(* POU FB_BACnet_RemoteProgram, ST *)
FUNCTION_BLOCK FB_BACnet_RemoteProgram
VAR_IN_OUT
	RemoteDevice		: FB_BACnet_RemoteDevice;
END_VAR
VAR_OUTPUT
	bReady				: BOOL;
	ePrgState			: E_BACNETPROGRAMSTATE;
	ePrgReasonHalt		: E_BACNETPROGRAMERROR;
	bOverridden			: BOOL;
	bOutOfService		: BOOL;
	bFault				: BOOL;
	bInAlarm			: BOOL;
	bError				: BOOL;
	nErrorId			: UINT;
END_VAR
VAR
	_ProgramState AT%I*: WORD;			(* ~(BACnet_ProgramState 				:		: )
								   			(BACnet_ObjectType 					: PROG	: )
			                            	(BACnet_RemoteCycletimeRead 		: 1000	: )
											(BACnet_RemoteFlagsRead        		: 1    	: )
                                   			(BACnet_RemoteResubscriptionInterval: 240 	: )
	                                		(BACnet_RemoteCycleTimeWrite   		: 1000	: )
	                                		(BACnet_RemoteFlagsWrite       		: 1		: )	*)
	_ReasonForHalt AT%I*: WORD;			(* ~(BACnet_ReasonForHalt 				: 		: )	*)
	_StatusFlags AT%I*: WORD;			(* ~(BACnet_StatusFlags 				:		: )	*)
	_nUpdateCount : UDINT := 0;
	_StatusFlagsBits : ST_BACnet_StatusFlags;
END_VAR
(* update client device *)
IF RemoteDevice._nUpdateCount = _nUpdateCount THEN
	RemoteDevice();
END_IF
(* remind current number of update counter *)
_nUpdateCount := RemoteDevice._nUpdateCount;

IF RemoteDevice.bFirstCycle THEN
	(* first call of the server device since reboot/reset *)
	bReady := FALSE;

ELSIF NOT RemoteDevice.bOperational THEN
	nErrorId := BACnet_ERR_OPERATIONAL;
	bReady := FALSE;

ELSIF _StatusFlags >= 4 THEN
	(* clear error flag *)
	nErrorId := BACnet_ERR_NO_ERROR;

	(* ready state *)
	bReady := TRUE;

	(* decode status flags *)
	_StatusFlagsBits := F_BACnet_StatusFlags(_StatusFlags);

	(* copy states to output *)
	bOverridden := _StatusFlagsBits.overridden;
	bOutOfService := _StatusFlagsBits.out_of_service;
	bFault := _StatusFlagsBits.fault;
	bInAlarm := _StatusFlagsBits.in_alarm;

	(* present value from BACnet *)
	ePrgState := _ProgramState;

	(* other states *)
	ePrgReasonHalt := _ReasonForHalt;
ELSE
	(* server device not ready, reset local ready also *)
	bReady := FALSE;
	(* and set error ID *)
	nErrorId := BACnet_ERR_WRONG_MAPPING;
END_IF

(* set error flag *)
bError := (nErrorId <> BACnet_ERR_NO_ERROR);
END_FUNCTION_BLOCK

(* POU FB_BACnet_RemoteProgram_EX, ST *)
FUNCTION_BLOCK FB_BACnet_RemoteProgram_EX
VAR_INPUT
	bEnablePV			: BOOL;
	ePV					: E_BACNETPROGRAMREQUEST;
	bRetrigger			: BOOL; (* execute selected request on raising edge again *)
END_VAR
VAR_IN_OUT
	RemoteDevice		: FB_BACnet_RemoteDevice;
END_VAR
VAR_OUTPUT
	bReady				: BOOL;
	ePrgState			: E_BACNETPROGRAMSTATE;
	ePrgChangeReq		: E_BACNETPROGRAMREQUEST;
	ePrgReasonHalt		: E_BACNETPROGRAMERROR;
	bOverridden			: BOOL;
	bOutOfService		: BOOL;
	bFault				: BOOL;
	bInAlarm			: BOOL;
	bProcessError		: BOOL;
	bOtherFault			: BOOL;
	tObjectID		: DINT := -1;
	bError				: BOOL;
	nErrorId			: UINT;
END_VAR
VAR
	_ProgramState AT%I*: WORD;			(* ~(BACnet_ProgramState 				:		: )
											(BACnet_ObjectType 					: PROG	: )
											(BACnet_RemoteCycletimeRead 		: 1000	: )
											(BACnet_RemoteFlagsRead        		: 1    	: )
											(BACnet_RemoteResubscriptionInterval: 240 	: )
											(BACnet_RemoteCycleTimeWrite   		: 1000	: )
											(BACnet_RemoteFlagsWrite       		: 1		: )	*)
	_ProgramChangeState AT%I*: WORD;	(* ~(BACnet_ProgramChange 				:		: )	*)
	_ReasonForHalt AT%I*: WORD;			(* ~(BACnet_ReasonForHalt 				: 		: )	*)
	_StatusFlags AT%I*: WORD;			(* ~(BACnet_StatusFlags 				:		: )	*)
	_Reliability AT%I*: WORD;			(* ~(BACnet_Reliability 				:		: )	*)
	_ProgramChangeRequest AT%Q*: WORD;	(* ~(BACnet_ProgramChange 				:		: )	*)
	_ObjectId AT%I*: DWORD;				(* ~(BACnet_ObjectIdentifier			:		: LINK) *)
	_nUpdateCount : UDINT := 0;
	_StatusFlagsBits : ST_BACnet_StatusFlags;
	_rtrigRetriggerPv : R_TRIG;
END_VAR
(* update client device *)
IF RemoteDevice._nUpdateCount = _nUpdateCount THEN
	RemoteDevice();
END_IF
(* remind current number of update counter *)
_nUpdateCount := RemoteDevice._nUpdateCount;

(* call trigger *)
_rtrigRetriggerPv(CLK:= bRetrigger, Q=> );

IF RemoteDevice.bFirstCycle THEN
	(* first call of the server device since reboot/reset *)
	bReady := FALSE;
	_ProgramChangeRequest := 0;
ELSIF NOT RemoteDevice.bOperational THEN
	nErrorId := BACnet_ERR_OPERATIONAL;
	bReady := FALSE;

ELSIF (F_BACnet_GetObjType(_ObjectId) <> BACnetObjectType_Program) THEN
	(* wrong mapping / invalid object ID *)
	IF _ObjectId = 0 THEN
		nErrorId := BACnet_ERR_WRONG_MAPPING;
	ELSE
		nErrorId := BACnet_ERR_INVALID_OBJECTID;
	END_IF
	bReady := FALSE;
	tObjectID := 16#FFFFFFFF;

ELSIF _StatusFlags >= 4 THEN
	(* clear error flag *)
	nErrorId := BACnet_ERR_NO_ERROR;

	(* ready state *)
	bReady := TRUE;

	(* decode status flags *)
	_StatusFlagsBits := F_BACnet_StatusFlags(_StatusFlags);

	(* copy states to output *)
	bOverridden := _StatusFlagsBits.overridden;
	bOutOfService := _StatusFlagsBits.out_of_service;
	bFault := _StatusFlagsBits.fault;
	bInAlarm := _StatusFlagsBits.in_alarm;
	bProcessError := (_Reliability = BACnetReliability_process_error);
	bOtherFault := (_Reliability = BACnetReliability_unreliable_other);
	tObjectID := _ObjectId;

	(* present value from BACnet *)
	ePrgState := _ProgramState;
	(* present value to BACnet *)
	IF bEnablePV THEN
		IF _rtrigRetriggerPv.Q THEN
			(* trigger request *)
			_ProgramChangeRequest := 0;
		ELSE
			(* set request value *)
			_ProgramChangeRequest := ePV;
		END_IF
	ELSE
		_ProgramChangeRequest := 0;
	END_IF
	(* other states *)
	ePrgReasonHalt := _ReasonForHalt;
	ePrgChangeReq := _ProgramChangeState;

ELSE
	(* server device not ready, reset local ready also *)
	bReady := FALSE;
	(* and set error ID *)
	nErrorId := BACnet_ERR_WRONG_MAPPING;
END_IF

(* set error flag *)
bError := (nErrorId <> BACnet_ERR_NO_ERROR);
END_FUNCTION_BLOCK

(* POU FB_BACnet_RemoteProgram_WR, ST *)
FUNCTION_BLOCK FB_BACnet_RemoteProgram_WR
VAR_INPUT
	bEnablePV			: BOOL;
	ePV					: E_BACNETPROGRAMREQUEST;
	bRetrigger			: BOOL; (* execute selected request on raising edge again *)
END_VAR
VAR_IN_OUT
	RemoteDevice		: FB_BACnet_RemoteDevice;
END_VAR
VAR_OUTPUT
	bReady				: BOOL;
	ePrgState			: E_BACNETPROGRAMSTATE;
	ePrgReasonHalt		: E_BACNETPROGRAMERROR;
	bOverridden			: BOOL;
	bOutOfService		: BOOL;
	bFault				: BOOL;
	bInAlarm			: BOOL;
	bError				: BOOL;
	nErrorId			: UINT;
END_VAR
VAR
	_ProgramState AT%I*: WORD;			(* ~(BACnet_ProgramState 				:		: )
								   			(BACnet_ObjectType 					: PROG	: )
			                            	(BACnet_RemoteCycletimeRead 		: 1000	: )
											(BACnet_RemoteFlagsRead        		: 1    	: )
                                   			(BACnet_RemoteResubscriptionInterval: 240 	: )
	                                		(BACnet_RemoteCycleTimeWrite   		: 1000	: )
	                                		(BACnet_RemoteFlagsWrite       		: 1		: )	*)
	_ReasonForHalt AT%I*: WORD;			(* ~(BACnet_ReasonForHalt 				: 		: )	*)
	_StatusFlags AT%I*: WORD;			(* ~(BACnet_StatusFlags 				:		: )	*)
	_ProgramChangeRequest AT%Q*: WORD;	(* ~(BACnet_ProgramChange 				:		: )	*)
	_nUpdateCount : UDINT := 0;
	_StatusFlagsBits : ST_BACnet_StatusFlags;
	_rtrigRetriggerPv : R_TRIG;
END_VAR
(* update client device *)
IF RemoteDevice._nUpdateCount = _nUpdateCount THEN
	RemoteDevice();
END_IF
(* remind current number of update counter *)
_nUpdateCount := RemoteDevice._nUpdateCount;

(* call trigger *)
_rtrigRetriggerPv(CLK:= bRetrigger, Q=> );

IF RemoteDevice.bFirstCycle THEN
	(* first call of the server device since reboot/reset *)
	bReady := FALSE;
	_ProgramChangeRequest := 0;
ELSIF NOT RemoteDevice.bOperational THEN
	nErrorId := BACnet_ERR_OPERATIONAL;
	bReady := FALSE;

ELSIF _StatusFlags >= 4 THEN
	(* clear error flag *)
	nErrorId := BACnet_ERR_NO_ERROR;

	(* ready state *)
	bReady := TRUE;

	(* decode status flags *)
	_StatusFlagsBits := F_BACnet_StatusFlags(_StatusFlags);

	(* copy states to output *)
	bOverridden := _StatusFlagsBits.overridden;
	bOutOfService := _StatusFlagsBits.out_of_service;
	bFault := _StatusFlagsBits.fault;
	bInAlarm := _StatusFlagsBits.in_alarm;

	(* present value from BACnet *)
	ePrgState := _ProgramState;
	(* present value to BACnet *)
	IF bEnablePV THEN
		IF _rtrigRetriggerPv.Q THEN
			(* trigger request *)
			_ProgramChangeRequest := 0;
		ELSE
			(* set request value *)
			_ProgramChangeRequest := ePV;
		END_IF
	ELSE
		_ProgramChangeRequest := 0;
	END_IF
	(* other states *)
	ePrgReasonHalt := _ReasonForHalt;
ELSE
	(* server device not ready, reset local ready also *)
	bReady := FALSE;
	(* and set error ID *)
	nErrorId := BACnet_ERR_WRONG_MAPPING;
END_IF

(* set error flag *)
bError := (nErrorId <> BACnet_ERR_NO_ERROR);
END_FUNCTION_BLOCK

(* POU FB_BACnet_RemotePulseConverter, ST *)
FUNCTION_BLOCK FB_BACnet_RemotePulseConverter
VAR_IN_OUT
	RemoteDevice		: FB_BACnet_RemoteDevice;
END_VAR
VAR_OUTPUT
	bReady				: BOOL;
	bOverridden			: BOOL;
	bOutOfService		: BOOL;
	bFault				: BOOL;
	bInAlarm			: BOOL;
	bError				: BOOL;
	nErrorId			: UINT;
END_VAR
VAR
	_StatusFlags AT%I*: UINT;		(* ~(BACnet_StatusFlags 				:		: )
										(BACnet_ObjectType 					: PC	: )
										(BACnet_RemoteCycletimeRead 		: 1000	: )
										(BACnet_RemoteFlagsRead        		: 1		: )
										(BACnet_RemoteResubscriptionInterval: 240	: )
                                		(BACnet_RemoteCycleTimeWrite   		: 1000	: )
                                		(BACnet_RemoteFlagsWrite       		: 1		: )	*)
	_StatusFlagsBits : ST_BACnet_StatusFlags;
	_nUpdateCount : UDINT := 0;
END_VAR
(* update client device *)
IF RemoteDevice._nUpdateCount = _nUpdateCount THEN
	RemoteDevice();
END_IF
(* remind current number of update counter *)
_nUpdateCount := RemoteDevice._nUpdateCount;

IF NOT RemoteDevice.bOperational THEN
	nErrorId := BACnet_ERR_OPERATIONAL;
	bReady := FALSE;

ELSIF _StatusFlags >= 4 THEN
	(* clear error flag *)
	nErrorId := BACnet_ERR_NO_ERROR;
	(* ready state *)
	bReady := TRUE;

	(* build bit states *)
	_StatusFlagsBits := F_BACnet_StatusFlags(_StatusFlags);

	(* copy states to output *)
	bOverridden := _StatusFlagsBits.overridden;
	bOutOfService := _StatusFlagsBits.out_of_service;
	bFault := _StatusFlagsBits.fault;
	bInAlarm := _StatusFlagsBits.in_alarm;

ELSE
	(* server device not ready, reset local ready also *)
	bReady := FALSE;
	(* and set error ID *)
	nErrorId := BACnet_ERR_WRONG_MAPPING;
END_IF

(* set error flag *)
bError := (nErrorId <> BACnet_ERR_NO_ERROR);
END_FUNCTION_BLOCK

(* POU FB_BACnet_RemotePulseConverter_EX, ST *)
FUNCTION_BLOCK FB_BACnet_RemotePulseConverter_EX
VAR_IN_OUT
	RemoteDevice	: FB_BACnet_RemoteDevice;
END_VAR
VAR_OUTPUT
	bReady			: BOOL;
	fPresentValue	: REAL;
	nCount			: UDINT;
	bOverridden		: BOOL;
	bOutOfService	: BOOL;
	bFault			: BOOL;
	bInAlarm		: BOOL;
	bOverRange		: BOOL;
	bUnderRange		: BOOL;
	bNoSensor		: BOOL;
	bOpenLoop		: BOOL;
	bShortedLoop	: BOOL;
	bCommFailure	: BOOL;
	bConfigError	: BOOL;
	bOtherFault		: BOOL;
	tObjectID		: T_BACnet_ObjectIdentifier := 16#FFFFFFFF;
	bError			: BOOL;
	nErrorId		: UINT;
END_VAR
VAR
	_ObjectId AT%I*: DWORD;		(* ~(BACnet_ObjectIdentifier			:		: LINK) *)
	_Count AT%I*: UDINT;		(* ~(BACnet_Count		 				:		: ) *)
	_PresentValue AT%I*: REAL;	(* ~(BACnet_PresentValue 				:		: )	*)
	_StatusFlags AT%I*: UINT;	(* ~(BACnet_StatusFlags 				:		: )
									(BACnet_ObjectType 					: PC	: )
									(BACnet_RemoteCycletimeRead 		: 1000	: )
									(BACnet_RemoteFlagsRead        		: 1		: )
									(BACnet_RemoteResubscriptionInterval: 240	: )
                                	(BACnet_RemoteCycleTimeWrite   		: 1000	: )
                                	(BACnet_RemoteFlagsWrite       		: 1		: )	*)
	_Reliability AT%I*:WORD;	(* ~(BACnet_Reliability					:		: )	*)
	_StatusFlagsBits : ST_BACnet_StatusFlags;
	_nUpdateCount : UDINT := 0;
END_VAR
(* update client device *)
IF RemoteDevice._nUpdateCount = _nUpdateCount THEN
	RemoteDevice();
END_IF
(* remind current number of update counter *)
_nUpdateCount := RemoteDevice._nUpdateCount;

IF NOT RemoteDevice.bOperational THEN
	nErrorId := BACnet_ERR_OPERATIONAL;
	bReady := FALSE;

ELSIF (F_BACnet_GetObjType(_ObjectId) <> BACnetObjectType_PulseConverter) THEN
	(* wrong mapping / invalid object ID *)
	IF _ObjectId = 0 THEN
		nErrorId := BACnet_ERR_WRONG_MAPPING;
	ELSE
		nErrorId := BACnet_ERR_INVALID_OBJECTID;
	END_IF
	bReady := FALSE;
	tObjectID := 16#FFFFFFFF;

ELSIF _StatusFlags >= 4 THEN
	(* clear error flag *)
	nErrorId := BACnet_ERR_NO_ERROR;
	(* ready state *)
	bReady := TRUE;

	(* present value *)
	fPresentValue := _PresentValue;
	nCount := _Count;

	(* build bit states *)
	_StatusFlagsBits := F_BACnet_StatusFlags(_StatusFlags);

	(* copy states to output *)
	bOverridden := _StatusFlagsBits.overridden;
	bOutOfService := _StatusFlagsBits.out_of_service;
	bFault := _StatusFlagsBits.fault;
	bInAlarm := _StatusFlagsBits.in_alarm;
	tObjectID := _ObjectId;

	(* reliability *)
	bOverRange	:= (_Reliability = BACnetReliability_over_range);
	bUnderRange	:= (_Reliability = BACnetReliability_under_range);
	bNoSensor	:= (_Reliability = BACnetReliability_no_sensor);
	bOpenLoop	:= (_Reliability = BACnetReliability_open_loop);
	bShortedLoop:= (_Reliability = BACnetReliability_shorted_loop);
	bCommFailure := (_Reliability = BACnetReliability_communication_failure);
	bConfigError:= (_Reliability = BACnetReliability_configuration_error);
	bOtherFault	:= (_Reliability = BACnetReliability_unreliable_other);

ELSE
	(* server device not ready, reset local ready also *)
	bReady := FALSE;
	(* and set error ID *)
	nErrorId := BACnet_ERR_WRONG_MAPPING;
END_IF

(* set error flag *)
bError := (nErrorId <> BACnet_ERR_NO_ERROR);
END_FUNCTION_BLOCK

(* POU FB_BACnet_RemoteSchedule, ST *)
FUNCTION_BLOCK FB_BACnet_RemoteSchedule
VAR_IN_OUT
	RemoteDevice			: FB_BACnet_RemoteDevice;
END_VAR
VAR_OUTPUT
	bReady				: BOOL;
	bPresentValue		: BOOL;
	bOverridden			: BOOL;
	bOutOfService		: BOOL;
	bFault				: BOOL;
	bInAlarm			: BOOL;
	bError				: BOOL;
	nErrorId			: UINT;
END_VAR
VAR
	_StatusFlags AT%I*: WORD; 	(* ~(BACnet_StatusFlags 				:		: )	*)
	_PresentValue AT%I*: BOOL;	(* ~(BACnet_PresentValueBool 			:		: )
									(BACnet_ObjectType 					: SCHED	: )
									(BACnet_RemoteCycletimeRead 		: 1000	: )
									(BACnet_RemoteFlagsRead        		: 1		: )
									(BACnet_RemoteResubscriptionInterval: 240	: )
                            		(BACnet_RemoteCycleTimeWrite   		: 1000	: )
                            		(BACnet_RemoteFlagsWrite       		: 1		: )	*)
	_StatusFlagsBits : ST_BACnet_StatusFlags;
	_nUpdateCount : UDINT := 0;
END_VAR
(* update client device *)
IF RemoteDevice._nUpdateCount = _nUpdateCount THEN
	RemoteDevice();
END_IF
(* remind current number of update counter *)
_nUpdateCount := RemoteDevice._nUpdateCount;

IF NOT RemoteDevice.bOperational THEN
	nErrorId := BACnet_ERR_OPERATIONAL;
	bReady := FALSE;

ELSIF _StatusFlags >= 4 THEN
	(* clear error flag *)
	nErrorId := BACnet_ERR_NO_ERROR;
	(* ready state *)
	bReady := TRUE;

	(* present value *)
	bPresentValue := _PresentValue;

	(* build bit states *)
	_StatusFlagsBits := F_BACnet_StatusFlags(_StatusFlags);

	(* copy states to output *)
	bOverridden := _StatusFlagsBits.overridden;
	bOutOfService := _StatusFlagsBits.out_of_service;
	bFault := _StatusFlagsBits.fault;
	bInAlarm := _StatusFlagsBits.in_alarm;

ELSE
	bReady := FALSE;
	(* and set error ID *)
	nErrorId := BACnet_ERR_WRONG_MAPPING;
END_IF

(* set error flag *)
bError := (nErrorId <> BACnet_ERR_NO_ERROR);
END_FUNCTION_BLOCK

(* POU FB_BACnet_RemoteSchedule_EX, ST *)
FUNCTION_BLOCK FB_BACnet_RemoteSchedule_EX
VAR_IN_OUT
	RemoteDevice			: FB_BACnet_RemoteDevice;
END_VAR
VAR_OUTPUT
	bReady				: BOOL;
	bPresentValue		: BOOL;
	bOverridden			: BOOL;
	bOutOfService		: BOOL;
	bFault				: BOOL;
	bInAlarm			: BOOL;
	bConfigError		: BOOL;
	bOtherFault			: BOOL;
	tObjectID			: T_BACnet_ObjectIdentifier := 16#FFFFFFFF;
	bError				: BOOL;
	nErrorId			: UINT;
END_VAR
VAR
	_ObjectId AT%I*: DWORD;				(* ~(BACnet_ObjectIdentifier			:		: LINK) *)
	_Reliability AT%I*: WORD; 			(* ~(BACnet_Reliability 				:		: )	*)
	_StatusFlags AT%I*: WORD; 			(* ~(BACnet_StatusFlags 				:		: )	*)
	_PresentValue AT%I*: BOOL;			(* ~(BACnet_PresentValueBool 			:		: )
											(BACnet_ObjectType 					: SCHED	: )
											(BACnet_RemoteCycletimeRead 		: 1000	: )
											(BACnet_RemoteFlagsRead        		: 1		: )
											(BACnet_RemoteResubscriptionInterval: 240	: )
                            				(BACnet_RemoteCycleTimeWrite   		: 1000	: )
                            				(BACnet_RemoteFlagsWrite       		: 1		: )	*)
	_StatusFlagsBits : ST_BACnet_StatusFlags;
	_nUpdateCount : UDINT := 0;
END_VAR
(* update client device *)
IF RemoteDevice._nUpdateCount = _nUpdateCount THEN
	RemoteDevice();
END_IF
(* remind current number of update counter *)
_nUpdateCount := RemoteDevice._nUpdateCount;

IF NOT RemoteDevice.bOperational THEN
	nErrorId := BACnet_ERR_OPERATIONAL;
	bReady := FALSE;

ELSIF (F_BACnet_GetObjType(_ObjectId) <> BACnetObjectType_Schedule) THEN
	(* wrong mapping / invalid object ID *)
	IF _ObjectId = 0 THEN
		nErrorId := BACnet_ERR_WRONG_MAPPING;
	ELSE
		nErrorId := BACnet_ERR_INVALID_OBJECTID;
	END_IF
	bReady := FALSE;
	tObjectID := 16#FFFFFFFF;

ELSIF _StatusFlags >= 4 THEN
	(* clear error flag *)
	nErrorId := BACnet_ERR_NO_ERROR;
	(* ready state *)
	bReady := TRUE;

	(* present value *)
	bPresentValue := _PresentValue;

	(* build bit states *)
	_StatusFlagsBits := F_BACnet_StatusFlags(_StatusFlags);

	(* copy states to output *)
	bOverridden := _StatusFlagsBits.overridden;
	bOutOfService := _StatusFlagsBits.out_of_service;
	bFault := _StatusFlagsBits.fault;
	bInAlarm := _StatusFlagsBits.in_alarm;
	bConfigError := (_Reliability = BACnetReliability_configuration_error);
	bOtherFault := (_Reliability = BACnetReliability_unreliable_other);
	tObjectID := _ObjectId;

ELSE
	bReady := FALSE;
	(* and set error ID *)
	nErrorId := BACnet_ERR_WRONG_MAPPING;
END_IF

(* set error flag *)
bError := (nErrorId <> BACnet_ERR_NO_ERROR);
END_FUNCTION_BLOCK

(* POU FB_BACnet_RemoteTrendLog, ST *)
FUNCTION_BLOCK FB_BACnet_RemoteTrendLog
VAR_IN_OUT
	RemoteDevice			: FB_BACnet_RemoteDevice;
END_VAR
VAR_OUTPUT
	bReady				: BOOL;
	bLogEnable			: BOOL;
	nRecordCount		: UDINT;
	nTotalCount			: UDINT;
	bError				: BOOL;
	nErrorId			: UINT;
END_VAR
VAR
	_RecordCount AT%I*: UDINT;		(* ~(BACnet_RecordCount					:		: )
										(BACnet_ObjectType					: TLOG	: )
										(BACnet_RemoteCycletimeRead 		: 1000	: )
										(BACnet_RemoteFlagsRead        		: 1		: )
										(BACnet_RemoteResubscriptionInterval: 240	: )
                                		(BACnet_RemoteCycleTimeWrite   		: 1000	: )
                                		(BACnet_RemoteFlagsWrite       		: 1		: )	*)
	_TotalRecordCount AT%I*: UDINT;	(* ~(BACnet_TotalRecordCount			:		: )	*)
	_LogEnable AT%I*: BOOL;			(* ~(BACnet_LogEnable					: 		: )	*)
	_nUpdateCount : UDINT := 0;
END_VAR
(* update client device *)
IF RemoteDevice._nUpdateCount = _nUpdateCount THEN
	RemoteDevice();
END_IF
(* remind current number of update counter *)
_nUpdateCount := RemoteDevice._nUpdateCount;

IF RemoteDevice.bOperational THEN
	(* clear error flag *)
	nErrorId := BACnet_ERR_NO_ERROR;
	(* ready state *)
	bReady := TRUE;

	(* other states *)
	nRecordCount := _RecordCount;
	nTotalCount := _TotalRecordCount;
	bLogEnable := _LogEnable;

ELSE
	bReady := FALSE;
	(* and set error ID *)
	nErrorId := BACnet_ERR_OPERATIONAL;
END_IF

(* set error flag *)
bError := (nErrorId <> BACnet_ERR_NO_ERROR);
END_FUNCTION_BLOCK

(* POU FB_BACnet_RemoteTrendLog_EX, ST *)
FUNCTION_BLOCK FB_BACnet_RemoteTrendLog_EX
VAR_OUTPUT
	bReady				: BOOL;
	bLogEnable			: BOOL;
	nRecordCount		: UDINT;
	nTotalCount			: UDINT;
	eEventState			: E_BACNETEVENTSTATE;
	tObjectID			: T_BACnet_ObjectIdentifier := 16#FFFFFFFF;
	bError				: BOOL;
	nErrorId			: UINT;
END_VAR
VAR_IN_OUT
	RemoteDevice			: FB_BACnet_RemoteDevice;
END_VAR
VAR
	_RecordCount AT%I*: UDINT;			(* ~(BACnet_RecordCount					:		: )
											(BACnet_ObjectType					: TLOG	: )
											(BACnet_RemoteCycletimeRead 		: 1000	: )
											(BACnet_RemoteFlagsRead        		: 1		: )
											(BACnet_RemoteResubscriptionInterval: 240	: )
											(BACnet_RemoteCycleTimeWrite   		: 1000	: )
                                			(BACnet_RemoteFlagsWrite       		: 1		: )	*)
	_TotalRecordCount AT%I*: UDINT;		(* ~(BACnet_TotalRecordCount			:		: )	*)
	_ObjectId AT%I*: DWORD;				(* ~(BACnet_ObjectIdentifier			:		: LINK) *)
	_EventState AT%I*: WORD;			(* ~(BACnet_EventState					:		: )	*)
	_LogEnable AT%I*: BOOL;				(* ~(BACnet_LogEnable					: 		: )	*)
	_nUpdateCount : UDINT := 0;
END_VAR
(* update client device *)
IF RemoteDevice._nUpdateCount = _nUpdateCount THEN
	RemoteDevice();
END_IF
(* remind current number of update counter *)
_nUpdateCount := RemoteDevice._nUpdateCount;

IF NOT RemoteDevice.bOperational THEN
	(* mapping seems to be wrong *)
	nErrorId := BACnet_ERR_OPERATIONAL;
	bReady := FALSE;

ELSIF (F_BACnet_GetObjType(_ObjectId) <> BACnetObjectType_TrendLog) THEN
	(* wrong mapping / invalid object ID *)
	IF _ObjectId = 0 THEN
		nErrorId := BACnet_ERR_WRONG_MAPPING;
	ELSE
		nErrorId := BACnet_ERR_INVALID_OBJECTID;
	END_IF
	bReady := FALSE;
	tObjectID := 16#FFFFFFFF;

ELSIF _EventState >= 0 THEN
	(* clear error flag *)
	nErrorId := BACnet_ERR_NO_ERROR;
	(* ready state *)
	bReady := TRUE;

	(* convert enumeration *)
	eEventState := _EventState;

	(* other states *)
	nRecordCount := _RecordCount;
	nTotalCount := _TotalRecordCount;
	bLogEnable := _LogEnable;
	tObjectID := _ObjectId;

ELSE
	bReady := FALSE;
	(* and set error ID *)
	nErrorId := BACnet_ERR_WRONG_MAPPING;
END_IF

(* set error flag *)
bError := (nErrorId <> BACnet_ERR_NO_ERROR);
END_FUNCTION_BLOCK

(* POU FB_BACnet_RemoteTrendLogMultiple, ST *)
FUNCTION_BLOCK FB_BACnet_RemoteTrendLogMultiple
VAR_IN_OUT
	RemoteDevice			: FB_BACnet_RemoteDevice;
END_VAR
VAR_OUTPUT
	bReady				: BOOL;
	bLogEnable			: BOOL;
	nRecordCount		: UDINT;
	nTotalCount			: UDINT;
	bError				: BOOL;
	nErrorId			: UINT;
END_VAR
VAR
	_RecordCount AT%I*: UDINT;		(* ~(BACnet_RecordCount					:		: )
										(BACnet_ObjectType					: TLM	: )
										(BACnet_RemoteCycletimeRead 		: 1000	: )
										(BACnet_RemoteFlagsRead        		: 1		: )
										(BACnet_RemoteResubscriptionInterval: 240	: )
                                		(BACnet_RemoteCycleTimeWrite   		: 1000	: )
                                		(BACnet_RemoteFlagsWrite       		: 1		: )	*)
	_TotalRecordCount AT%I*: UDINT;	(* ~(BACnet_TotalRecordCount			:		: )	*)
	_LogEnable AT%I*: BOOL;			(* ~(BACnet_LogEnable					: 		: )	*)
	_nUpdateCount : UDINT := 0;
END_VAR
(* update client device *)
IF RemoteDevice._nUpdateCount = _nUpdateCount THEN
	RemoteDevice();
END_IF
(* remind current number of update counter *)
_nUpdateCount := RemoteDevice._nUpdateCount;

IF RemoteDevice.bOperational THEN
	(* clear error flag *)
	nErrorId := BACnet_ERR_NO_ERROR;
	(* ready state *)
	bReady := TRUE;

	(* other states *)
	nRecordCount := _RecordCount;
	nTotalCount := _TotalRecordCount;
	bLogEnable := _LogEnable;

ELSE
	bReady := FALSE;
	(* and set error ID *)
	nErrorId := BACnet_ERR_OPERATIONAL;
END_IF

(* set error flag *)
bError := (nErrorId <> BACnet_ERR_NO_ERROR);
END_FUNCTION_BLOCK

(* POU FB_BACnet_RemoteTrendLogMultiple_EX, ST *)
FUNCTION_BLOCK FB_BACnet_RemoteTrendLogMultiple_EX
VAR_OUTPUT
	bReady				: BOOL;
	bLogEnable			: BOOL;
	nRecordCount		: UDINT;
	nTotalCount			: UDINT;
	eEventState			: E_BACNETEVENTSTATE;
	tObjectID			: T_BACnet_ObjectIdentifier := 16#FFFFFFFF;
	bError				: BOOL;
	nErrorId			: UINT;
END_VAR
VAR_IN_OUT
	RemoteDevice			: FB_BACnet_RemoteDevice;
END_VAR
VAR
	_RecordCount AT%I*: UDINT;			(* ~(BACnet_RecordCount					:		: )
											(BACnet_ObjectType					: TLM	: )
											(BACnet_RemoteCycletimeRead 		: 1000	: )
											(BACnet_RemoteFlagsRead        		: 1		: )
											(BACnet_RemoteResubscriptionInterval: 240	: )
											(BACnet_RemoteCycleTimeWrite   		: 1000	: )
                                			(BACnet_RemoteFlagsWrite       		: 1		: )	*)
	_TotalRecordCount AT%I*: UDINT;		(* ~(BACnet_TotalRecordCount			:		: )	*)
	_ObjectId AT%I*: DWORD;				(* ~(BACnet_ObjectIdentifier			:		: LINK) *)
	_EventState AT%I*: WORD;			(* ~(BACnet_EventState					:		: )	*)
	_LogEnable AT%I*: BOOL;				(* ~(BACnet_LogEnable					: 		: )	*)
	_nUpdateCount : UDINT := 0;
END_VAR
(* update client device *)
IF RemoteDevice._nUpdateCount = _nUpdateCount THEN
	RemoteDevice();
END_IF
(* remind current number of update counter *)
_nUpdateCount := RemoteDevice._nUpdateCount;

IF NOT RemoteDevice.bOperational THEN
	(* mapping seems to be wrong *)
	nErrorId := BACnet_ERR_OPERATIONAL;
	bReady := FALSE;

ELSIF (F_BACnet_GetObjType(_ObjectId) <> BACnetObjectType_TrendLogMultiple) THEN
	(* wrong mapping / invalid object ID *)
	IF _ObjectId = 0 THEN
		nErrorId := BACnet_ERR_WRONG_MAPPING;
	ELSE
		nErrorId := BACnet_ERR_INVALID_OBJECTID;
	END_IF
	bReady := FALSE;
	tObjectID := 16#FFFFFFFF;

ELSIF _EventState >= 0 THEN
	(* clear error flag *)
	nErrorId := BACnet_ERR_NO_ERROR;
	(* ready state *)
	bReady := TRUE;

	(* convert enumeration *)
	eEventState := _EventState;

	(* other states *)
	nRecordCount := _RecordCount;
	nTotalCount := _TotalRecordCount;
	bLogEnable := _LogEnable;
	tObjectID := _ObjectId;

ELSE
	bReady := FALSE;
	(* and set error ID *)
	nErrorId := BACnet_ERR_WRONG_MAPPING;
END_IF

(* set error flag *)
bError := (nErrorId <> BACnet_ERR_NO_ERROR);
END_FUNCTION_BLOCK

(* POU FB_BACnet_Schedule, ST *)
FUNCTION_BLOCK FB_BACnet_Schedule
VAR_IN_OUT
	Device	: FB_BACnet_Device;
END_VAR
VAR_OUTPUT
	bReady			: BOOL;
	bPresentValue	: BOOL;
	bOverridden		: BOOL;
	bOutOfService	: BOOL;
	bFault			: BOOL;
	bInAlarm		: BOOL;
	bError			: BOOL;
	nErrorId		: UINT;
END_VAR
VAR
	_StatusFlags AT%I*: WORD; 	(* ~(BACnet_StatusFlags 				:		: )	*)
	_PresentValue AT%I*: BOOL;	(* ~(BACnet_PresentValueBool 			:		: )
									(BACnet_ObjectType 					: SCHED	: )	*)
	_StatusFlagsBits : ST_BACnet_StatusFlags;
	_nUpdateCount : UDINT := 0;
END_VAR
(* update server device *)
IF (Device._nUpdateCount = _nUpdateCount) THEN
	Device();
END_IF
(* remind current number of update counter *)
_nUpdateCount := Device._nUpdateCount;

(* check BitString format of StatusFlags --> if StatusFlags are less than 4, object isn't linked correctly *)
IF (_StatusFlags < 4) THEN
	(* wrong mapping *)
	nErrorId := BACnet_ERR_WRONG_MAPPING;
	bReady := FALSE;

ELSIF Device.bOperational THEN
	(* ready state *)
	bReady := TRUE;
	nErrorId := BACnet_ERR_NO_ERROR;

	(* present value *)
	bPresentValue := _PresentValue;

	(* build bit states *)
	_StatusFlagsBits := F_BACnet_StatusFlags(_StatusFlags);

	(* copy states to output *)
	bOverridden := _StatusFlagsBits.overridden;
	bOutOfService := _StatusFlagsBits.out_of_service;
	bFault := _StatusFlagsBits.fault;
	bInAlarm := _StatusFlagsBits.in_alarm;

ELSE
	bReady := FALSE;
	nErrorId := BACnet_ERR_OPERATIONAL;
END_IF
(* set error flag *)
bError := (nErrorId <> BACnet_ERR_NO_ERROR);
END_FUNCTION_BLOCK

(* POU FB_BACnet_Schedule_EX, ST *)
FUNCTION_BLOCK FB_BACnet_Schedule_EX
VAR_IN_OUT
	Device				: FB_BACnet_Device;
END_VAR
VAR_OUTPUT
	bReady				: BOOL;
	bPresentValue		: BOOL;
	bOverridden			: BOOL;
	bOutOfService		: BOOL;
	bFault				: BOOL;
	bInAlarm			: BOOL;
	bConfigError		: BOOL;
	bOtherFault			: BOOL;
	tObjectID			: T_BACnet_ObjectIdentifier := 16#FFFFFFFF;
	bError				: BOOL;
	nErrorId			: UINT;
END_VAR
VAR
	_ObjectId AT%I*: DWORD;		(* ~(BACnet_ObjectIdentifier		:		: LINK) *)
	_Reliability AT%I*: WORD; 	(* ~(BACnet_Reliability 			:		: )	*)
	_StatusFlags AT%I*: WORD; 	(* ~(BACnet_StatusFlags 			:		: )	*)
	_PresentValue AT%I*: BOOL;	(* ~(BACnet_PresentValueBool 		:		: )
									(BACnet_ObjectType 				: SCHED	: )	*)
	_StatusFlagsBits : ST_BACnet_StatusFlags;
	_nUpdateCount : UDINT := 0;
END_VAR
(* update server device *)
IF (Device._nUpdateCount = _nUpdateCount) THEN
	Device();
END_IF
(* remind current number of update counter *)
_nUpdateCount := Device._nUpdateCount;

(* check object type *)
IF (F_BACnet_GetObjType(_ObjectId) <> BACnetObjectType_Schedule) THEN
	(* wrong mapping / invalid object ID *)
	IF _ObjectId = 0 THEN
		nErrorId := BACnet_ERR_WRONG_MAPPING;
	ELSE
		nErrorId := BACnet_ERR_INVALID_OBJECTID;
	END_IF
	bReady := FALSE;

ELSIF (_StatusFlags < 4) THEN
	(* wrong mapping *)
	nErrorId := BACnet_ERR_WRONG_MAPPING;
	bReady := FALSE;

ELSIF Device.bOperational THEN
	(* ready state *)
	bReady := TRUE;
	nErrorId := BACnet_ERR_NO_ERROR;

	(* present value *)
	bPresentValue := _PresentValue;

	(* build bit states *)
	_StatusFlagsBits := F_BACnet_StatusFlags(_StatusFlags);

	(* copy states to output *)
	bOverridden := _StatusFlagsBits.overridden;
	bOutOfService := _StatusFlagsBits.out_of_service;
	bFault := _StatusFlagsBits.fault;
	bInAlarm := _StatusFlagsBits.in_alarm;
	bConfigError := (_Reliability = BACnetReliability_configuration_error);
	bOtherFault := (_Reliability = BACnetReliability_unreliable_other);
	tObjectID := _ObjectId;

ELSE
	bReady := FALSE;
	nErrorId := BACnet_ERR_OPERATIONAL;
END_IF
(* set error flag *)
bError := (nErrorId <> BACnet_ERR_NO_ERROR);
END_FUNCTION_BLOCK

(* POU FB_BACnet_TimeSync, ST *)
FUNCTION_BLOCK FB_BACnet_TimeSync
VAR_INPUT
	bExecute	: BOOL; (* Synchronize BACnet time information with local system time and, if set, send broadcast message *)
	bBroadcast	: BOOL := TRUE; (* Synchronize BACnet with broadcast message (FALSE = No broadcast [Rev-12-only feature]) *)
	tTimeout	: TIME := BACnet_ADSTimeOut;
END_VAR
VAR_IN_OUT
	Device		: FB_BACnet_Device;
END_VAR
VAR_OUTPUT
	bReady		: BOOL; (* local time information is valid *)
	bBusy		: BOOL;
	bError		: BOOL;
	nErrID		: UDINT;
	tsSystemTime: TIMESTRUCT; (* local system time (windows time) as TIMESTRUCT *)
	dtSystemTime: ST_BACnet_DateTime; (* local system time (windows time) as BACnet_Date_Time *)
	tzID		: E_TimeZoneID;
	tzInfo		: ST_TimeZoneInformation;
	tsUTC		: TIMESTRUCT; (* UTC system time (GMT) *)
END_VAR
VAR
	_fbAdsWrite	: ADSWRITE;
	_fbLocalTime: FB_LocalSystemTime;
	_fbGetTzInfo: FB_GetTimeZoneInformation;
	_fbUTC		: FB_TzSpecificLocalTimeToSystemTime;
	_oldTzId	: E_TimeZoneID := eTimeZoneID_Invalid;
	_tofReload	: TOF;
	_dtUTC		: ST_BACnet_DateTime;
END_VAR
(* read local time *)
_fbLocalTime(
	sNetID	:= '',
	bEnable	:= TRUE,
	dwCycle	:= ,
	dwOpt	:= ,
	tTimeout:= tTimeout,
	bValid	=> ,
	systemTime=> tsSystemTime,
	tzID	=> );

_fbGetTzInfo(
	sNetID	:= '',
	bExecute:= _fbLocalTime.bValid AND (_oldTzId <> _fbLocalTime.tzID) AND (NOT _tofReload.Q),
	tTimeout:= tTimeout,
	bBusy	=> ,
	bError	=> ,
	nErrID	=> ,
	tzID	=> ,
	tzInfo	=> tzInfo);

_tofReload(
	IN	:= _fbGetTzInfo.bError AND (NOT _tofReload.Q),
	PT	:= tTimeout,
	Q	=> ,
	ET	=> );

IF _fbGetTzInfo.bExecute AND (NOT _fbGetTzInfo.bBusy) THEN
	IF (NOT _fbGetTzInfo.bError) THEN
		_oldTzId := _fbLocalTime.tzID;
	ELSE
		_oldTzId := eTimeZoneID_Invalid;
	END_IF
END_IF

_fbUTC(
	in		:= _fbLocalTime.systemTime,
	tzInfo	:= _fbGetTzInfo.tzInfo,
	out		=> tsUTC,
	eTzID	=> tzID,
	bB		=> );

(* check if all information are valid *)
bReady := _fbLocalTime.bValid AND (NOT _fbGetTzInfo.bError) AND (_fbUTC.eTzID > eTimeZoneID_Unknown) AND Device.stAdsConn.bValid;

(* convert to BACnet_Date_Time *)
dtSystemTime:= F_BACnet_TimeStruct_TO_DateTime(tsSystemTime);
_dtUTC		:= F_BACnet_TimeStruct_TO_DateTime(tsUTC);

(* call ADS write function to synchronize system time *)
IF bBroadcast THEN
	_fbAdsWrite.IDXOFFS	:= 16#0000;
ELSE
	_fbAdsWrite.IDXOFFS	:= 16#0001;
END_IF
_fbAdsWrite(
	NETID	:= Device.stAdsConn.sAmsNetId,
	PORT	:= 16#FFFF, (* AMS port of BACnet device adapter *)
	IDXGRP	:= 16#8000002D,
	LEN		:= SIZEOF(_dtUTC),
	SRCADDR	:= ADR(_dtUTC),
	WRITE	:= bReady AND bExecute,
	TMOUT	:= tTimeout,
	BUSY	=> bBusy,
	ERR		=> bError,
	ERRID	=> nErrID);
END_FUNCTION_BLOCK

(* POU FB_BACnet_TrendLog, ST *)
FUNCTION_BLOCK FB_BACnet_TrendLog
VAR_IN_OUT
	Device	: FB_BACnet_Device;
END_VAR
VAR_OUTPUT
	bReady			: BOOL;
	bLogEnable		: BOOL;
	nTotalCount		: UDINT;
	bError			: BOOL;
	nErrorId		: UINT;
END_VAR
VAR
	_TotalRecordCount AT%I*: UDINT;	(* ~(BACnet_TotalRecordCount:		: )
										(BACnet_ObjectType		: TLOG	: )	*)
	_LogEnable AT%I*: BOOL;			(* ~(BACnet_LogEnable		: 		: )	*)
	_nUpdateCount : UDINT := 0;
END_VAR
(* update server device *)
IF (Device._nUpdateCount = _nUpdateCount) THEN
	Device();
END_IF
(* remind current number of update counter *)
_nUpdateCount := Device._nUpdateCount;

IF Device.bOperational THEN
	(* ready state *)
	bReady := TRUE;
	nErrorId := BACnet_ERR_NO_ERROR;
	bLogEnable := _LogEnable;

	(* other states *)
	nTotalCount := _TotalRecordCount;

ELSE
	bReady := FALSE;
	nErrorId := BACnet_ERR_OPERATIONAL;
END_IF
(* set error flag *)
bError := (nErrorId <> BACnet_ERR_NO_ERROR);
END_FUNCTION_BLOCK

(* POU FB_BACnet_TrendLog_EX, ST *)
FUNCTION_BLOCK FB_BACnet_TrendLog_EX
VAR_IN_OUT
	Device	: FB_BACnet_Device;
END_VAR
VAR_OUTPUT
	bReady			: BOOL;
	bLogEnable		: BOOL;
	nRecordCount	: UDINT;
	nTotalCount		: UDINT;
	eEventState		: E_BACNETEVENTSTATE;
	bAckedTrans_ToOffNormal : BOOL;
	bAckedTrans_ToFault		: BOOL;
	bAckedTrans_ToNormal	: BOOL;
	tObjectID		: DINT := -1;
	bError			: BOOL;
	nErrorId		: UINT;
END_VAR
VAR
	_RecordCount AT%I*: UDINT;		(* ~(BACnet_RecordCount			:		: )
										(BACnet_ObjectType			: TLOG	: )	*)
	_TotalRecordCount AT%I*: UDINT;	(* ~(BACnet_TotalRecordCount	:		: )	*)
	_ObjectId AT%I*: DWORD;			(* ~(BACnet_ObjectIdentifier	:		: LINK) *)
	_EventState AT%I*: WORD;		(* ~(BACnet_EventState			:		: )	*)
	_AckedTransitions AT%I*:WORD;	(* ~(BACnet_AckedTransitions	:		: ) *)
	_LogEnable AT%I*: BOOL;			(* ~(BACnet_LogEnable			: 		: )	*)
	_AckedTransBits : ST_BACnet_EventTransitionBits;
	_nUpdateCount : UDINT := 0;
END_VAR
(* update server device *)
IF (Device._nUpdateCount = _nUpdateCount) THEN
	Device();
END_IF
(* remind current number of update counter *)
_nUpdateCount := Device._nUpdateCount;

(* check object type *)
IF (F_BACnet_GetObjType(_ObjectId) <> BACnetObjectType_TrendLog) THEN
	(* wrong mapping / invalid object ID *)
	IF _ObjectId = 0 THEN
		nErrorId := BACnet_ERR_WRONG_MAPPING;
	ELSE
		nErrorId := BACnet_ERR_INVALID_OBJECTID;
	END_IF
	bReady := FALSE;

ELSIF Device.bOperational THEN
	(* ready state *)
	bReady := TRUE;
	bLogEnable := _LogEnable;
	nErrorId := BACnet_ERR_NO_ERROR;

	(* build bit states *)
	_AckedTransBits		:= F_BACnet_EventTransitionFlags(_AckedTransitions);
	bAckedTrans_ToOffNormal := _AckedTransBits.to_offnormal;
	bAckedTrans_ToFault := _AckedTransBits.to_fault;
	bAckedTrans_ToNormal := _AckedTransBits.to_normal;
	tObjectID := _ObjectId;

	(* convert enumeration *)
	eEventState := _EventState;

	(* other states *)
	nRecordCount := _RecordCount;
	nTotalCount := _TotalRecordCount;

ELSE
	bReady := FALSE;
	nErrorId := BACnet_ERR_OPERATIONAL;
END_IF
(* set error flag *)
bError := (nErrorId <> BACnet_ERR_NO_ERROR);
END_FUNCTION_BLOCK

(* POU FB_BACnet_TrendLogMultiple, ST *)
FUNCTION_BLOCK FB_BACnet_TrendLogMultiple
VAR_IN_OUT
	Device	: FB_BACnet_Device;
END_VAR
VAR_OUTPUT
	bReady			: BOOL;
	bLogEnable		: BOOL;
	nTotalCount		: UDINT;
	bError			: BOOL;
	nErrorId		: UINT;
END_VAR
VAR
	_TotalRecordCount AT%I*: UDINT;	(* ~(BACnet_TotalRecordCount:		: )
										(BACnet_ObjectType		: TLM	: )	*)
	_LogEnable AT%I*: BOOL;			(* ~(BACnet_LogEnable		: 		: )	*)
	_nUpdateCount : UDINT := 0;
END_VAR
(* update server device *)
IF (Device._nUpdateCount = _nUpdateCount) THEN
	Device();
END_IF
(* remind current number of update counter *)
_nUpdateCount := Device._nUpdateCount;

IF Device.bOperational THEN
	(* ready state *)
	bReady := TRUE;
	nErrorId := BACnet_ERR_NO_ERROR;
	bLogEnable := _LogEnable;

	(* other states *)
	nTotalCount := _TotalRecordCount;

ELSE
	bReady := FALSE;
	nErrorId := BACnet_ERR_OPERATIONAL;
END_IF
(* set error flag *)
bError := (nErrorId <> BACnet_ERR_NO_ERROR);
END_FUNCTION_BLOCK

(* POU FB_BACnet_TrendLogMultiple_EX, ST *)
FUNCTION_BLOCK FB_BACnet_TrendLogMultiple_EX
VAR_IN_OUT
	Device	: FB_BACnet_Device;
END_VAR
VAR_OUTPUT
	bReady			: BOOL;
	bLogEnable		: BOOL;
	nRecordCount	: UDINT;
	nTotalCount		: UDINT;
	eEventState		: E_BACNETEVENTSTATE;
	bAckedTrans_ToOffNormal : BOOL;
	bAckedTrans_ToFault		: BOOL;
	bAckedTrans_ToNormal	: BOOL;
	tObjectID		: DINT := -1;
	bError			: BOOL;
	nErrorId		: UINT;
END_VAR
VAR
	_RecordCount AT%I*: UDINT;		(* ~(BACnet_RecordCount			:		: )
										(BACnet_ObjectType			: TLM	: )	*)
	_TotalRecordCount AT%I*: UDINT;	(* ~(BACnet_TotalRecordCount	:		: )	*)
	_ObjectId AT%I*: DWORD;			(* ~(BACnet_ObjectIdentifier	:		: LINK) *)
	_EventState AT%I*: WORD;		(* ~(BACnet_EventState			:		: )	*)
	_AckedTransitions AT%I*:WORD;	(* ~(BACnet_AckedTransitions	:		: ) *)
	_LogEnable AT%I*: BOOL;			(* ~(BACnet_LogEnable			: 		: )	*)
	_AckedTransBits : ST_BACnet_EventTransitionBits;
	_nUpdateCount : UDINT := 0;
END_VAR
(* update server device *)
IF (Device._nUpdateCount = _nUpdateCount) THEN
	Device();
END_IF
(* remind current number of update counter *)
_nUpdateCount := Device._nUpdateCount;

(* check object type *)
IF (F_BACnet_GetObjType(_ObjectId) <> BACnetObjectType_TrendLogMultiple) THEN
	(* wrong mapping / invalid object ID *)
	IF _ObjectId = 0 THEN
		nErrorId := BACnet_ERR_WRONG_MAPPING;
	ELSE
		nErrorId := BACnet_ERR_INVALID_OBJECTID;
	END_IF
	bReady := FALSE;

ELSIF Device.bOperational THEN
	(* ready state *)
	bReady := TRUE;
	bLogEnable := _LogEnable;
	nErrorId := BACnet_ERR_NO_ERROR;

	(* build bit states *)
	_AckedTransBits		:= F_BACnet_EventTransitionFlags(_AckedTransitions);
	bAckedTrans_ToOffNormal := _AckedTransBits.to_offnormal;
	bAckedTrans_ToFault := _AckedTransBits.to_fault;
	bAckedTrans_ToNormal := _AckedTransBits.to_normal;
	tObjectID := _ObjectId;

	(* convert enumeration *)
	eEventState := _EventState;

	(* other states *)
	nRecordCount := _RecordCount;
	nTotalCount := _TotalRecordCount;

ELSE
	bReady := FALSE;
	nErrorId := BACnet_ERR_OPERATIONAL;
END_IF
(* set error flag *)
bError := (nErrorId <> BACnet_ERR_NO_ERROR);
END_FUNCTION_BLOCK

(* POU FB_BACnet_WeeklyScheduleProperty, ST *)
FUNCTION_BLOCK FB_BACnet_WeeklyScheduleProperty
VAR_INPUT
	tObjectID			: T_BACnet_ObjectIdentifier := 16#FFFFFFFF;
	bAutoGet			: BOOL:=TRUE; (* TRUE = get data from property when ADS connection OR object ID changed *)
	bGet				: BOOL; (* FALSE --> TRUE = get data from property *)
	bSet				: BOOL; (* FALSE --> TRUE = set data into property *)
END_VAR
VAR_IN_OUT
	stWeeklySched		: ST_BACnet_WeeklyScheduleBool;
	stAdsConn			: ST_BACnet_AdsConnection;
END_VAR
VAR_OUTPUT
	bDone				: BOOL;
	bBusy				: BOOL;
	bError				: BOOL;
	nErrorId			: UINT;
END_VAR
VAR
	_fbReadProp		: FB_BACnet_ReadProp;
	_fbWriteProp	: FB_BACnet_WriteProp;
	_i				: INT;
	_pDailySched	: POINTER TO ST_BACnet_DailySchedule;
	_pTimeValue		: POINTER TO ST_BACnet_TimeValueList;
	_pOldTimeValue	: POINTER TO ST_BACnet_TimeValueList;
	_iDayBuffer		: INT;
	_iDayEntryBuf	: INT;
	_rtrigGet		: R_TRIG;
	_rtrigSet		: R_TRIG;

	_cbTmpSize		: UDINT;
	_cbTotalEntry	: UDINT;
	_cbTotalBuf		: UDINT;
	_bNextDay		: BOOL;
	_bNextTimeValue	: BOOL;
	_nDays			: UINT;
	_nAdsReloadOld	: USINT;
	_tObjectIDOld	: T_BACnet_ObjectIdentifier := 16#FFFFFFFF;

END_VAR
(*

Listheader:

typedef struct _ListEntryHdr
{
      DWORD nEntrySize;
      DWORD hdrInfo;
}ListEntryHdr, *PListEntryHdr;

#define ListAlignedSize(n)         (4*(((n)+3)/4))
#define FirstListEntry(p) ( (p)->nEntrySize == 0 )                          ? NULL:p
#define NextListEntry(p) ( ( ((p)->nEntrySize&0x80000000) == 0 ) ? NULL:(PBYTE)(p) + ( ListAlignedSize((p)->nEntrySize&~(0x80000000)) + sizeof(ListEntryHdr)) ) // +4 da für nEntrySize 4 Byte reserviert sind, HighBit ausmaskieren
#define ElemSize(p) ((p)->nEntrySize&(~0x80000000))
#define AlignedEntrySize(p) (ListAlignedSize((p)->nEntrySize&(~0x80000000)))

###################################################################

PropExceptionSchedule:

enum BACnetSpecialEventChoice
{
      calendarEntry,
      calendarReference,
      MaxBACnetSpecialEventChoice
};

typedef struct _BACnetCalendarEntry
{
      BACnetCalendarEntryChoice choice;
      union
      {
            BACnetDate              date;
            BACnetDateRange   dateRange;
            BACnetWeekNDay          weekNDay;
      };
}BACnetCalendarEntry, *PBACnetCalendarEntry;

enum BACnetValueChoice
{
      NullValue                    = 0,
      BoolValue                    = 1,
      UnsignedValue                = 2,
      SignedValue                  = 3,
      RealValue                    = 4,
      DoubleValue                  = 5,
      OctedStringValue        = 6,
      CharStringValue         = 7,
      ObjectIdentifierValue = 8,   // but DataType is 0x0C
      EnumerationValue        = 9,
      MaxBACnetValueChoice    = 10
};

typedef struct _BACnetValue  
{
      BACnetValueChoice choice;
      DWORD                        length;     // Alignment + Datenlänge die folgt
      union
      {
            BOOL                                     boolValue;
            FLOAT                                    realValue;
            DOUBLE                                   doubleValue;
            INT                                      signedValue;
            UINT                                     unsignedValue;
            BYTE*                                    pOctedStringValue; 
            CHAR*                                    pCharStringValue;
            BACnetObjectIdentifier  objectIdentifierValue;
            EnumerationValueType         enumerationValue;
      };
}BACnetValue, *PBACnetValue;

typedef struct _BACnetTimeValue
{
      BACnetTime time;
      DWORD  reserved;  // 64bit Alignment
      BACnetValue value;
}BACnetTimeValue, *PBACnetTimeValue;

typedef struct _BACnetTimeValueList
{
      DWORD nEntrySize; // 0x80000000 -> next entry
      DWORD reserved;
      BACnetTimeValue listEntry;
}BACnetTimeValueList, *PBACnetTimeValueList;

typedef struct _BACnetSpecialEvent
{
      BACnetSpecialEventChoice choice;
      union
      {
            BACnetCalendarEntry calendarEntry;
            BACnetObjectIdentifier calendarReference;
      };
      DWORD eventPriority; // DWORD due to alignment
      DWORD reserved;
      BACnetTimeValueList listOfTimeValues;
}BACnetSpecialEvent, *PBACnetSpecialEvent;

typedef struct _BACnetSpecialEventList
{
      DWORD nEntrySize; // 0x80000000 -> next entry
      DWORD reserved;
      BACnetSpecialEvent listEntry;
}BACnetSpecialEventList, *PBACnetSpecialEventList;

###################################################################

PropWeeklySchedule:

typedef struct _BACnetDailySchedule
{
      DWORD nEntrySize; // 0x80000000 -> next entry
      DWORD reserved;
      BACnetTimeValueList listEntry;
} BACnetDailySchedule, *PBACnetDailySchedule;

###################################################################

PropScheduleDefault / PropPresentValue

typedef struct _BACnetValueList
{
      DWORD nEntrySize; // 0x80000000 -> next entry
      DWORD reserved;
      BACnetValue listEntry;
} BACnetValueList, *PBACnetValueList;

###################################################################

*)

(* ADS read *)
_fbReadProp(
	BACnetDevicePort	:= stAdsConn.nAmsPort,
	bExecute			:= ,
	sNetId				:= stAdsConn.sAmsNetId,
	ObjectType			:= F_BACnet_GetObjType(tObjectID),
	PropertyID			:= BACnetPropertyIdentifier_WeeklySchedule,
	DataType			:= BACnetDataType_DailyScheduleList,
	ObjectInstance		:= F_BACnet_GetObjInstance(tObjectID),
	ptrValue			:= ADR(stBACnet_AdsBuffer.arrData),
	nLenValue			:= SIZEOF(stBACnet_AdsBuffer.arrData),
	bDone				=> ,
	bBusy				=> ,
	bError				=> ,
	nErrID				=> ,
	nProcessedLen		=> );

_fbWriteProp(
	BACnetDevicePort	:= stAdsConn.nAmsPort,
	bExecute			:= ,
	sNetId				:= stAdsConn.sAmsNetId,
	ObjectType			:= F_BACnet_GetObjType(tObjectID),
	PropertyID			:= BACnetPropertyIdentifier_WeeklySchedule,
	Priority			:= BACnetPriority_None,
	DataType			:= BACnetDataType_DailyScheduleList,
	ObjectInstance		:= F_BACnet_GetObjInstance(tObjectID),
	ptrValue			:= ADR(stBACnet_AdsBuffer.arrData),
	nLenValue			:= _cbTotalBuf,
	bDone				=> ,
	bBusy				=> ,
	bError				=> ,
	nErrID				=> );

(* trigger start event *)
_rtrigGet(CLK:= bGet, Q=> );
_rtrigSet(CLK:= bSet, Q=> );

(* state machine *)
CASE _i OF

	0: (* Idle *)
		IF 		_rtrigGet.Q
			OR	_rtrigSet.Q
			OR	(		(		(_nAdsReloadOld <> stAdsConn.nReload)
							OR	(_tObjectIDOld <> tObjectID)
						)
					AND	bAutoGet
				)
			OR	stWeeklySched.bReqGet
			OR	stWeeklySched.bReqSet
		THEN
			IF (NOT stAdsConn.bValid) THEN
				(* ADS connection not valid *)
				nErrorId := BACnet_ERR_INVALID_ADS_CONN;
			ELSIF (NOT stAdsConn.bServer AND NOT stAdsConn.bClient) THEN
				(* not a server nor a client *)
				nErrorId := BACnet_ERR_ADS_NoServerClient;
			ELSE
				(* check day count *)
				_nDays := SIZEOF(stWeeklySched.arrEntries) / SIZEOF(stWeeklySched.arrEntries[0]);
				(* decide get or set *)
				IF _rtrigGet.Q OR stWeeklySched.bReqGet THEN
					_i := 1;
					stWeeklySched.bReqGet := FALSE;
				ELSIF _rtrigSet.Q OR stWeeklySched.bReqSet THEN
					_i := 11;
					stWeeklySched.bReqSet := FALSE;
				ELSIF bAutoGet THEN
					_i := 1;
					stWeeklySched.bReqGet := FALSE;
				END_IF
				nErrorId := BACnet_ERR_NO_ERROR;
				(* remind parameter *)
				_tObjectIDOld := tObjectID;
				_nAdsReloadOld := stAdsConn.nReload;
				(* lock data array *)
				stWeeklySched.bBusy := TRUE;
			END_IF
			(* reset done flag *)
			bDone := FALSE;
		END_IF
		IF (NOT bGet) AND (NOT bSet) AND (NOT bAutoGet) THEN
			nErrorId := BACnet_ERR_NO_ERROR;
			bDone := FALSE;
		END_IF

	(* READ *)
	1: (* read object property data over ADS *)
		IF TestAndSet(stBACnet_AdsBuffer.bTestSet) THEN
			IF _fbReadProp.bExecute THEN
				IF _fbReadProp.bError THEN
					_i := 100;
					nErrorId := BACnet_ERR_ADS_Read;
					_fbReadProp.bExecute := FALSE;
				ELSIF (NOT _fbReadProp.bBusy) THEN
					_i := 2;
					_fbReadProp.bExecute := FALSE;
					_pDailySched := ADR(stBACnet_AdsBuffer.arrData);
					MEMSET(ADR(stWeeklySched.arrEntries), 0, SIZEOF(stWeeklySched.arrEntries));
					_iDayBuffer := 0;
					_cbTotalBuf := 0;
				END_IF
			ELSE
				(* lock global ADS buffer and start reading *)
				IF stBACnet_AdsBuffer.iLocked = 0 THEN
					_fbReadProp.bExecute := TRUE;
					stBACnet_AdsBuffer.iLocked := SIZEOF(stBACnet_AdsBuffer.arrData);
				END_IF
			END_IF

			(* release temporary task lock *)
			stBACnet_AdsBuffer.bTestSet := FALSE;
		END_IF

	2: (* select day *)
		_pTimeValue := ADR(_pDailySched^.stListEntry);
		(* scan time value list *)
		_iDayEntryBuf := 0;
		_i := 3;

	3: (* select time value *)
		WHILE (_i = 3) DO
			(* check entry size of time value *)
			IF (_pTimeValue^.nEntrySize AND 16#7FFFFFFF) > 0 THEN
				(* check internal schedule buffer index *)
				IF (_iDayBuffer > _nDays-1) THEN
					(* error, wrong day index *)
					nErrorId := BACnet_ERR_ADS_SchedData;
					_i := 100;
				ELSE
					IF (_iDayEntryBuf <= BACnet_MaxDayEntry) THEN
						IF _pTimeValue^.stListEntry.stValue.eValueChoice = BACnetDataType_Null THEN
							(* NULL *)
							stWeeklySched.arrEntries[_iDayBuffer][_iDayEntryBuf].stTime	:= _pTimeValue^.stListEntry.stTime;
							stWeeklySched.arrEntries[_iDayBuffer][_iDayEntryBuf].eType		:= _pTimeValue^.stListEntry.stValue.eValueChoice;
							stWeeklySched.arrEntries[_iDayBuffer][_iDayEntryBuf].bValue	:= FALSE;
							stWeeklySched.arrEntries[_iDayBuffer][_iDayEntryBuf].bValid	:= TRUE;
							_iDayEntryBuf := _iDayEntryBuf + 1;

						ELSIF (_pTimeValue^.stListEntry.stValue.cbData = 1) THEN
							(* read time, data type and value *)
							stWeeklySched.arrEntries[_iDayBuffer][_iDayEntryBuf].stTime	:= _pTimeValue^.stListEntry.stTime;
							stWeeklySched.arrEntries[_iDayBuffer][_iDayEntryBuf].eType		:= _pTimeValue^.stListEntry.stValue.eValueChoice;
							stWeeklySched.arrEntries[_iDayBuffer][_iDayEntryBuf].bValue	:= FALSE;
							MEMCPY(	ADR(stWeeklySched.arrEntries[_iDayBuffer][_iDayEntryBuf].bValue),
									ADR(_pTimeValue^.stListEntry.stValue.nData),
									MIN(	SIZEOF(stWeeklySched.arrEntries[_iDayBuffer][_iDayEntryBuf].bValue),
											_pTimeValue^.stListEntry.stValue.cbData
										)
							);
							stWeeklySched.arrEntries[_iDayBuffer][_iDayEntryBuf].bValid	:= TRUE;
							_iDayEntryBuf := _iDayEntryBuf + 1;
						ELSE
							(* unsupported data type length *);
						END_IF
					END_IF

					(* next time value entry *)
					_NextTimeValue();
					(* check if next time value entry available *)
					IF (NOT _bNextTimeValue) THEN
						(* update pointer each cycle (even if no day follows!) *)
						_NextDay();
						(* check for next day *)
						IF _bNextDay THEN
							(* go on *)
							_iDayBuffer := _iDayBuffer + 1;
							_i := 2;
						ELSE
							(* DONE *)
							_i := 4;
						END_IF
					END_IF
				END_IF

			ELSE
				(* update pointer each cycle (even if no day follows!) *)
				_NextDay();
				(* No timevalue entry, check if next day element exists and pointer is plausible *)
				IF _bNextDay THEN
					(* next day entry exists, go on *)
					_iDayBuffer := _iDayBuffer + 1;
					(* check pointer *)
					IF (_pDailySched + (_pDailySched^.nEntrySize AND 16#7FFFFFFF)) < (ADR(stBACnet_AdsBuffer.arrData) + SIZEOF(stBACnet_AdsBuffer.arrData)) THEN
						_i := 2;
					ELSE
						(* buffer too small *)
						nErrorId := BACnet_ERR_ADS_BufferSize;
						_i := 100;
					END_IF
				ELSE
					(* DONE *)
					_i := 4;
				END_IF
			END_IF
		END_WHILE

	4: (* data read and parsed successful *)
		stWeeklySched.nGet := stWeeklySched.nGet +1;
		_i := 100;

	(* WRITE *)
	11: (* lock global ADS buffer *)
		IF TestAndSet(stBACnet_AdsBuffer.bTestSet) THEN
			IF stBACnet_AdsBuffer.iLocked = 0 THEN
				stBACnet_AdsBuffer.iLocked := SIZEOF(stBACnet_AdsBuffer.arrData);
				_i := 12;
				(*MEMSET(ADR(stBACnet_AdsBuffer.arrData), 0, SIZEOF(stBACnet_AdsBuffer.arrData));*)
			END_IF
			(* release temporary task lock *)
			stBACnet_AdsBuffer.bTestSet := FALSE;
		END_IF

	12: (* prepare data *)
		(* set day pointer *)
		_pDailySched := ADR(stBACnet_AdsBuffer.arrData);
		_cbTotalBuf := 0;
		(* scan schedule data *)
		FOR _iDayBuffer := 0 TO _nDays-1 DO
			(* set timevalue pointer *)
			_pTimeValue := ADR(_pDailySched^.stListEntry);
			_cbTotalEntry := 0;
			_pOldTimeValue := 0;
			(* scan time values *)
			FOR _iDayEntryBuf := 0 TO BACnet_MaxDayEntry DO
				IF		stWeeklySched.arrEntries[_iDayBuffer][_iDayEntryBuf].bValid
					AND	(		stWeeklySched.arrEntries[_iDayBuffer][_iDayEntryBuf].eType = BACnetDataType_Bool
							OR	stWeeklySched.arrEntries[_iDayBuffer][_iDayEntryBuf].eType = BACnetDataType_Null
						)
				THEN
					(* set flag "next entry" to the previous element *)
					IF (_iDayEntryBuf > 0) AND (_pOldTimeValue <> 0) THEN
						_pOldTimeValue^.nEntrySize := _pOldTimeValue^.nEntrySize + 16#80000000;
					END_IF
					(* set data *)
					_pTimeValue^.stListEntry.stValue.nData := 0; (* clear data *)
					_pTimeValue^.stListEntry.stTime := stWeeklySched.arrEntries[_iDayBuffer][_iDayEntryBuf].stTime;
					(* decide between None and Bool type *)
					IF stWeeklySched.arrEntries[_iDayBuffer][_iDayEntryBuf].eType = BACnetDataType_Bool THEN
						_pTimeValue^.stListEntry.stValue.cbData := SIZEOF(stWeeklySched.arrEntries[_iDayBuffer][_iDayEntryBuf].bValue);
						_pTimeValue^.stListEntry.stValue.eValueChoice := BACnetDataType_Bool;
						_pTimeValue^.stListEntry.stValue.nRes1 := 0;
						MEMCPY(	ADR(_pTimeValue^.stListEntry.stValue.nData),
								ADR(stWeeklySched.arrEntries[_iDayBuffer][_iDayEntryBuf].bValue),
								1
						);
					ELSE
						(* unsupported *)
						_pTimeValue^.stListEntry.stValue.cbData := 0;
						_pTimeValue^.stListEntry.stValue.eValueChoice := BACnetDataType_Null;
						_pTimeValue^.stListEntry.stValue.nRes1 := 0;
					END_IF

					(* calculate time-value entry size *)
					_pTimeValue^.nEntrySize :=	_pTimeValue^.stListEntry.stValue.cbData
											+	SIZEOF(_pTimeValue^.stListEntry.nRes)
											+	SIZEOF(_pTimeValue^.stListEntry.stTime)
											+	SIZEOF(_pTimeValue^.stListEntry.stValue.cbData)
											+	SIZEOF(_pTimeValue^.stListEntry.stValue.eValueChoice)
											+	SIZEOF(_pTimeValue^.stListEntry.stValue.nRes1);

					(* update time value pointer *)
					_NextTimeValue();

					(* ...and add to total entry size counter *)
					_cbTotalEntry := _cbTotalEntry + _cbTmpSize;
				ELSE
					(* reset time value entry *)
					_pTimeValue^.nEntrySize := 0;
					_pTimeValue^.stListEntry.stValue.cbData := 0;
					_pTimeValue^.stListEntry.stValue.nRes1 := 0;
				END_IF
			END_FOR

			(* caclulate day-entry size *)
			_pDailySched^.nEntrySize := MAX(_cbTotalEntry, SIZEOF(_pDailySched^.stListEntry.nEntrySize) + SIZEOF(_pDailySched^.stListEntry.nRes));

			(* next day? *)
			IF (_iDayBuffer < _nDays-1) THEN
				_pDailySched^.nEntrySize := _pDailySched^.nEntrySize + 16#80000000;
			END_IF

			(* update pointer each cycle (even if no day follows!) *)
			_NextDay();
		END_FOR
		(* send data *)
		_i := 13;

	13:
		IF _fbWriteProp.bExecute AND (NOT _fbWriteProp.bBusy) THEN
			(* check result *)
			_fbWriteProp.bExecute := FALSE;
			IF _fbWriteProp.bError THEN
				nErrorId := BACnet_ERR_ADS_Write;
			ELSE
				stWeeklySched.nSet := stWeeklySched.nSet +1;
			END_IF
			_i := 100;
		ELSE
			(* start ADS write *)
			_fbWriteProp.bExecute := TRUE;
		END_IF

	100: (* Done *)
		bDone := (nErrorId = BACnet_ERR_NO_ERROR);
		(* release ADS buffer *)
		stBACnet_AdsBuffer.iLocked := 0;
		(* release data array *)
		stWeeklySched.bBusy := FALSE;
		(* go idle *)
		_i := 0;

END_CASE

(* set error flag *)
bError 	:= nErrorId > BACnet_ERR_NO_ERROR;
bBusy 	:= _i > 0;
END_FUNCTION_BLOCK
ACTION _NextDay:
_bNextDay := ((_pDailySched^.nEntrySize AND 16#80000000) = 16#80000000);
_cbTmpSize := _F_BACnet_AlignedSize(_pDailySched^.nEntrySize AND 16#7FFFFFFF) + SIZEOF(_pDailySched^.nEntrySize) + SIZEOF(_pDailySched^.nRes);
_pDailySched := _pDailySched + _cbTmpSize;
_cbTotalBuf := _cbTotalBuf + _cbTmpSize;
_pOldTimeValue := 0;
END_ACTION
ACTION _NextTimeValue:
_bNextTimeValue := (_pTimeValue^.nEntrySize AND 16#80000000) = 16#80000000;
_cbTmpSize := _F_BACnet_AlignedSize(_pTimeValue^.nEntrySize AND 16#7FFFFFFF) + SIZEOF(_pDailySched^.stListEntry.nEntrySize) + SIZEOF(_pDailySched^.stListEntry.nRes);
_pOldTimeValue := _pTimeValue;
_pTimeValue := _pTimeValue + _cbTmpSize;
END_ACTION

(* POU FB_BACnet_WeeklySchedulePropertyReal, ST *)
FUNCTION_BLOCK FB_BACnet_WeeklySchedulePropertyReal
VAR_INPUT
	tObjectID			: T_BACnet_ObjectIdentifier := 16#FFFFFFFF;
	bAutoGet			: BOOL:=TRUE; (* TRUE = get data from property when ADS connection OR object ID changed *)
	bGet				: BOOL; (* FALSE --> TRUE = get data from property *)
	bSet				: BOOL; (* FALSE --> TRUE = set data into property *)
END_VAR
VAR_IN_OUT
	stWeeklySched		: ST_BACnet_WeeklyScheduleReal;
	stAdsConn			: ST_BACnet_AdsConnection;
END_VAR
VAR_OUTPUT
	bDone				: BOOL;
	bBusy				: BOOL;
	bError				: BOOL;
	nErrorId			: UINT;
END_VAR
VAR
	_fbReadProp		: FB_BACnet_ReadProp;
	_fbWriteProp	: FB_BACnet_WriteProp;
	_i				: INT;
	_pDailySched	: POINTER TO ST_BACnet_DailySchedule;
	_pTimeValue		: POINTER TO ST_BACnet_TimeValueList;
	_pOldTimeValue	: POINTER TO ST_BACnet_TimeValueList;
	_iDayBuffer		: INT;
	_iDayEntryBuf	: INT;
	_rtrigGet		: R_TRIG;
	_rtrigSet		: R_TRIG;

	_cbTmpSize		: UDINT;
	_cbTotalEntry	: UDINT;
	_cbTotalBuf		: UDINT;
	_bNextDay		: BOOL;
	_bNextTimeValue	: BOOL;
	_nDays			: UINT;
	_nAdsReloadOld	: USINT;
	_tObjectIDOld	: T_BACnet_ObjectIdentifier := 16#FFFFFFFF;

	_pReal			: POINTER TO REAL;
END_VAR
(*

Listheader:

typedef struct _ListEntryHdr
{
      DWORD nEntrySize;
      DWORD hdrInfo;
}ListEntryHdr, *PListEntryHdr;

#define ListAlignedSize(n)         (4*(((n)+3)/4))
#define FirstListEntry(p) ( (p)->nEntrySize == 0 )                          ? NULL:p
#define NextListEntry(p) ( ( ((p)->nEntrySize&0x80000000) == 0 ) ? NULL:(PBYTE)(p) + ( ListAlignedSize((p)->nEntrySize&~(0x80000000)) + sizeof(ListEntryHdr)) ) // +4 da für nEntrySize 4 Byte reserviert sind, HighBit ausmaskieren
#define ElemSize(p) ((p)->nEntrySize&(~0x80000000))
#define AlignedEntrySize(p) (ListAlignedSize((p)->nEntrySize&(~0x80000000)))

###################################################################

PropExceptionSchedule:

enum BACnetSpecialEventChoice
{
      calendarEntry,
      calendarReference,
      MaxBACnetSpecialEventChoice
};

typedef struct _BACnetCalendarEntry
{
      BACnetCalendarEntryChoice choice;
      union
      {
            BACnetDate              date;
            BACnetDateRange   dateRange;
            BACnetWeekNDay          weekNDay;
      };
}BACnetCalendarEntry, *PBACnetCalendarEntry;

enum BACnetValueChoice
{
      NullValue                    = 0,
      BoolValue                    = 1,
      UnsignedValue                = 2,
      SignedValue                  = 3,
      RealValue                    = 4,
      DoubleValue                  = 5,
      OctedStringValue        = 6,
      CharStringValue         = 7,
      ObjectIdentifierValue = 8,   // but DataType is 0x0C
      EnumerationValue        = 9,
      MaxBACnetValueChoice    = 10
};

typedef struct _BACnetValue  
{
      BACnetValueChoice choice;
      DWORD                        length;     // Alignment + Datenlänge die folgt
      union
      {
            BOOL                                     boolValue;
            FLOAT                                    realValue;
            DOUBLE                                   doubleValue;
            INT                                      signedValue;
            UINT                                     unsignedValue;
            BYTE*                                    pOctedStringValue; 
            CHAR*                                    pCharStringValue;
            BACnetObjectIdentifier  objectIdentifierValue;
            EnumerationValueType         enumerationValue;
      };
}BACnetValue, *PBACnetValue;

typedef struct _BACnetTimeValue
{
      BACnetTime time;
      DWORD  reserved;  // 64bit Alignment
      BACnetValue value;
}BACnetTimeValue, *PBACnetTimeValue;

typedef struct _BACnetTimeValueList
{
      DWORD nEntrySize; // 0x80000000 -> next entry
      DWORD reserved;
      BACnetTimeValue listEntry;
}BACnetTimeValueList, *PBACnetTimeValueList;

typedef struct _BACnetSpecialEvent
{
      BACnetSpecialEventChoice choice;
      union
      {
            BACnetCalendarEntry calendarEntry;
            BACnetObjectIdentifier calendarReference;
      };
      DWORD eventPriority; // DWORD due to alignment
      DWORD reserved;
      BACnetTimeValueList listOfTimeValues;
}BACnetSpecialEvent, *PBACnetSpecialEvent;

typedef struct _BACnetSpecialEventList
{
      DWORD nEntrySize; // 0x80000000 -> next entry
      DWORD reserved;
      BACnetSpecialEvent listEntry;
}BACnetSpecialEventList, *PBACnetSpecialEventList;

###################################################################

PropWeeklySchedule:

typedef struct _BACnetDailySchedule
{
      DWORD nEntrySize; // 0x80000000 -> next entry
      DWORD reserved;
      BACnetTimeValueList listEntry;
} BACnetDailySchedule, *PBACnetDailySchedule;

###################################################################

PropScheduleDefault / PropPresentValue

typedef struct _BACnetValueList
{
      DWORD nEntrySize; // 0x80000000 -> next entry
      DWORD reserved;
      BACnetValue listEntry;
} BACnetValueList, *PBACnetValueList;

###################################################################

*)

(* ADS read *)
_fbReadProp(
	BACnetDevicePort	:= stAdsConn.nAmsPort,
	bExecute			:= ,
	sNetId				:= stAdsConn.sAmsNetId,
	ObjectType			:= F_BACnet_GetObjType(tObjectID),
	PropertyID			:= BACnetPropertyIdentifier_WeeklySchedule,
	DataType			:= BACnetDataType_DailyScheduleList,
	ObjectInstance		:= F_BACnet_GetObjInstance(tObjectID),
	ptrValue			:= ADR(stBACnet_AdsBuffer.arrData),
	nLenValue			:= SIZEOF(stBACnet_AdsBuffer.arrData),
	bDone				=> ,
	bBusy				=> ,
	bError				=> ,
	nErrID				=> ,
	nProcessedLen		=> );

_fbWriteProp(
	BACnetDevicePort	:= stAdsConn.nAmsPort,
	bExecute			:= ,
	sNetId				:= stAdsConn.sAmsNetId,
	ObjectType			:= F_BACnet_GetObjType(tObjectID),
	PropertyID			:= BACnetPropertyIdentifier_WeeklySchedule,
	Priority			:= BACnetPriority_None,
	DataType			:= BACnetDataType_DailyScheduleList,
	ObjectInstance		:= F_BACnet_GetObjInstance(tObjectID),
	ptrValue			:= ADR(stBACnet_AdsBuffer.arrData),
	nLenValue			:= _cbTotalBuf,
	bDone				=> ,
	bBusy				=> ,
	bError				=> ,
	nErrID				=> );

(* trigger start event *)
_rtrigGet(CLK:= bGet, Q=> );
_rtrigSet(CLK:= bSet, Q=> );

(* state machine *)
CASE _i OF

	0: (* Idle *)
		IF 		_rtrigGet.Q
			OR	_rtrigSet.Q
			OR	(		(		(_nAdsReloadOld <> stAdsConn.nReload)
							OR	(_tObjectIDOld <> tObjectID)
						)
					AND	bAutoGet
				)
			OR	stWeeklySched.bReqGet
			OR	stWeeklySched.bReqSet
		THEN
			IF (NOT stAdsConn.bValid) THEN
				(* ADS connection not valid *)
				nErrorId := BACnet_ERR_INVALID_ADS_CONN;
			ELSIF (NOT stAdsConn.bServer AND NOT stAdsConn.bClient) THEN
				(* not a server nor a client *)
				nErrorId := BACnet_ERR_ADS_NoServerClient;
			ELSE
				(* check day count *)
				_nDays := SIZEOF(stWeeklySched.arrEntries) / SIZEOF(stWeeklySched.arrEntries[0]);
				(* decide get or set *)
				IF _rtrigGet.Q OR stWeeklySched.bReqGet THEN
					_i := 1;
					stWeeklySched.bReqGet := FALSE;
				ELSIF _rtrigSet.Q OR stWeeklySched.bReqSet THEN
					_i := 11;
					stWeeklySched.bReqSet := FALSE;
				ELSIF bAutoGet THEN
					_i := 1;
					stWeeklySched.bReqGet := FALSE;
				END_IF
				nErrorId := BACnet_ERR_NO_ERROR;
				(* remind parameter *)
				_tObjectIDOld := tObjectID;
				_nAdsReloadOld := stAdsConn.nReload;
				(* lock data array *)
				stWeeklySched.bBusy := TRUE;
			END_IF
			(* reset done flag *)
			bDone := FALSE;
		END_IF
		IF (NOT bGet) AND (NOT bSet) AND (NOT bAutoGet) THEN
			nErrorId := BACnet_ERR_NO_ERROR;
			bDone := FALSE;
		END_IF

	(* READ *)
	1: (* read object property data over ADS *)
		IF TestAndSet(stBACnet_AdsBuffer.bTestSet) THEN
			IF _fbReadProp.bExecute THEN
				IF _fbReadProp.bError THEN
					_i := 100;
					nErrorId := BACnet_ERR_ADS_Read;
					_fbReadProp.bExecute := FALSE;
				ELSIF (NOT _fbReadProp.bBusy) THEN
					_i := 2;
					_fbReadProp.bExecute := FALSE;
					_pDailySched := ADR(stBACnet_AdsBuffer.arrData);
					MEMSET(ADR(stWeeklySched.arrEntries), 0, SIZEOF(stWeeklySched.arrEntries));
					_iDayBuffer := 0;
					_cbTotalBuf := 0;
				END_IF
			ELSE
				(* lock global ADS buffer and start reading *)
				IF stBACnet_AdsBuffer.iLocked = 0 THEN
					_fbReadProp.bExecute := TRUE;
					stBACnet_AdsBuffer.iLocked := SIZEOF(stBACnet_AdsBuffer.arrData);
				END_IF
			END_IF

			(* release temporary task lock *)
			stBACnet_AdsBuffer.bTestSet := FALSE;
		END_IF

	2: (* select day *)
		_pTimeValue := ADR(_pDailySched^.stListEntry);
		(* scan time value list *)
		_iDayEntryBuf := 0;
		_i := 3;

	3: (* select time value *)
		WHILE (_i = 3) DO
			(* check entry size of time value *)
			IF (_pTimeValue^.nEntrySize AND 16#7FFFFFFF) > 0 THEN
				(* check internal schedule buffer index *)
				IF (_iDayBuffer > _nDays-1) THEN
					(* error, wrong day index *)
					nErrorId := BACnet_ERR_ADS_SchedData;
					_i := 100;
				ELSE
					IF (_iDayEntryBuf <= BACnet_MaxDayEntry) THEN
						IF _pTimeValue^.stListEntry.stValue.eValueChoice = BACnetDataType_Null THEN
							(* NULL *)
							stWeeklySched.arrEntries[_iDayBuffer][_iDayEntryBuf].stTime	:= _pTimeValue^.stListEntry.stTime;
							stWeeklySched.arrEntries[_iDayBuffer][_iDayEntryBuf].eType		:= _pTimeValue^.stListEntry.stValue.eValueChoice;
							stWeeklySched.arrEntries[_iDayBuffer][_iDayEntryBuf].rValue	:= F_BACnet_NAN();
							stWeeklySched.arrEntries[_iDayBuffer][_iDayEntryBuf].bValid	:= TRUE;
							_iDayEntryBuf := _iDayEntryBuf + 1;

						ELSIF (_pTimeValue^.stListEntry.stValue.cbData = 4) THEN
							(* read time, data type and value *)
							stWeeklySched.arrEntries[_iDayBuffer][_iDayEntryBuf].stTime	:= _pTimeValue^.stListEntry.stTime;
							stWeeklySched.arrEntries[_iDayBuffer][_iDayEntryBuf].eType		:= _pTimeValue^.stListEntry.stValue.eValueChoice;
							stWeeklySched.arrEntries[_iDayBuffer][_iDayEntryBuf].rValue	:= F_BACnet_NAN();
							MEMCPY(	ADR(stWeeklySched.arrEntries[_iDayBuffer][_iDayEntryBuf].rValue),
									ADR(_pTimeValue^.stListEntry.stValue.nData),
									MIN(	SIZEOF(stWeeklySched.arrEntries[_iDayBuffer][_iDayEntryBuf].rValue),
											_pTimeValue^.stListEntry.stValue.cbData
										)
							);
							stWeeklySched.arrEntries[_iDayBuffer][_iDayEntryBuf].bValid	:= TRUE;
							_iDayEntryBuf := _iDayEntryBuf + 1;
						ELSE
							(* unsupported data type length *);
						END_IF
					END_IF

					(* next time value entry *)
					_NextTimeValue();
					(* check if next time value entry available *)
					IF (NOT _bNextTimeValue) THEN
						(* update pointer each cycle (even if no day follows!) *)
						_NextDay();
						(* check for next day *)
						IF _bNextDay THEN
							(* go on *)
							_iDayBuffer := _iDayBuffer + 1;
							_i := 2;
						ELSE
							(* DONE *)
							_i := 4;
						END_IF
					END_IF
				END_IF

			ELSE
				(* update pointer each cycle (even if no day follows!) *)
				_NextDay();
				(* No timevalue entry, check if next day element exists and pointer is plausible *)
				IF _bNextDay THEN
					(* next day entry exists, go on *)
					_iDayBuffer := _iDayBuffer + 1;
					(* check pointer *)
					IF (_pDailySched + (_pDailySched^.nEntrySize AND 16#7FFFFFFF)) < (ADR(stBACnet_AdsBuffer.arrData) + SIZEOF(stBACnet_AdsBuffer.arrData)) THEN
						_i := 2;
					ELSE
						(* buffer too small *)
						nErrorId := BACnet_ERR_ADS_BufferSize;
						_i := 100;
					END_IF
				ELSE
					(* DONE *)
					_i := 4;
				END_IF
			END_IF
		END_WHILE

	4: (* data read and parsed successful *)
		stWeeklySched.nGet := stWeeklySched.nGet +1;
		_i := 100;

	(* WRITE *)
	11: (* lock global ADS buffer *)
		IF TestAndSet(stBACnet_AdsBuffer.bTestSet) THEN
			IF stBACnet_AdsBuffer.iLocked = 0 THEN
				stBACnet_AdsBuffer.iLocked := SIZEOF(stBACnet_AdsBuffer.arrData);
				_i := 12;
				(*MEMSET(ADR(stBACnet_AdsBuffer.arrData), 0, SIZEOF(stBACnet_AdsBuffer.arrData));*)
			END_IF
			(* release temporary task lock *)
			stBACnet_AdsBuffer.bTestSet := FALSE;
		END_IF

	12: (* prepare data *)
		(* set day pointer *)
		_pDailySched := ADR(stBACnet_AdsBuffer.arrData);
		_cbTotalBuf := 0;
		(* scan schedule data *)
		FOR _iDayBuffer := 0 TO _nDays-1 DO
			(* set timevalue pointer *)
			_pTimeValue := ADR(_pDailySched^.stListEntry);
			_cbTotalEntry := 0;
			_pOldTimeValue := 0;
			(* scan time values *)
			FOR _iDayEntryBuf := 0 TO BACnet_MaxDayEntry DO
				IF		stWeeklySched.arrEntries[_iDayBuffer][_iDayEntryBuf].bValid
					AND	(		stWeeklySched.arrEntries[_iDayBuffer][_iDayEntryBuf].eType = BACnetDataType_Real
							OR	stWeeklySched.arrEntries[_iDayBuffer][_iDayEntryBuf].eType = BACnetDataType_Null
						)
				THEN
					(* set flag "next entry" to the previous element *)
					IF (_iDayEntryBuf > 0) AND (_pOldTimeValue <> 0) THEN
						_pOldTimeValue^.nEntrySize := _pOldTimeValue^.nEntrySize + 16#80000000;
					END_IF
					(* set data *)
					_pReal := ADR(_pTimeValue^.stListEntry.stValue.nData);
					_pReal^ := 0.0; (* clear data *)
					_pTimeValue^.stListEntry.stTime := stWeeklySched.arrEntries[_iDayBuffer][_iDayEntryBuf].stTime;
					(* decide between None and Real type *)
					IF stWeeklySched.arrEntries[_iDayBuffer][_iDayEntryBuf].eType = BACnetDataType_Real THEN
						_pTimeValue^.stListEntry.stValue.cbData := SIZEOF(stWeeklySched.arrEntries[_iDayBuffer][_iDayEntryBuf].rValue);
						_pTimeValue^.stListEntry.stValue.eValueChoice := BACnetDataType_Real;
						_pTimeValue^.stListEntry.stValue.nRes1 := 0;
						MEMCPY(	_pReal,
								ADR(stWeeklySched.arrEntries[_iDayBuffer][_iDayEntryBuf].rValue),
								4
						);
					ELSE
						(* unsupported *)
						_pTimeValue^.stListEntry.stValue.cbData := 0;
						_pTimeValue^.stListEntry.stValue.eValueChoice := BACnetDataType_Null;
						_pTimeValue^.stListEntry.stValue.nRes1 := 0;
					END_IF

					(* calculate time-value entry size *)
					_pTimeValue^.nEntrySize :=	_pTimeValue^.stListEntry.stValue.cbData
											+	SIZEOF(_pTimeValue^.stListEntry.nRes)
											+	SIZEOF(_pTimeValue^.stListEntry.stTime)
											+	SIZEOF(_pTimeValue^.stListEntry.stValue.cbData)
											+	SIZEOF(_pTimeValue^.stListEntry.stValue.eValueChoice)
											+	SIZEOF(_pTimeValue^.stListEntry.stValue.nRes1);

					(* update time value pointer *)
					_NextTimeValue();

					(* ...and add to total entry size counter *)
					_cbTotalEntry := _cbTotalEntry + _cbTmpSize;
				ELSE
					(* reset time value entry *)
					_pTimeValue^.nEntrySize := 0;
					_pTimeValue^.stListEntry.stValue.cbData := 0;
					_pTimeValue^.stListEntry.stValue.nRes1 := 0;
				END_IF
			END_FOR

			(* caclulate day-entry size *)
			_pDailySched^.nEntrySize := MAX(_cbTotalEntry, SIZEOF(_pDailySched^.stListEntry.nEntrySize) + SIZEOF(_pDailySched^.stListEntry.nRes));

			(* next day? *)
			IF (_iDayBuffer < _nDays-1) THEN
				_pDailySched^.nEntrySize := _pDailySched^.nEntrySize + 16#80000000;
			END_IF

			(* update pointer each cycle (even if no day follows!) *)
			_NextDay();
		END_FOR
		(* send data *)
		_i := 13;

	13:
		IF _fbWriteProp.bExecute AND (NOT _fbWriteProp.bBusy) THEN
			(* check result *)
			_fbWriteProp.bExecute := FALSE;
			IF _fbWriteProp.bError THEN
				nErrorId := BACnet_ERR_ADS_Write;
			ELSE
				stWeeklySched.nSet := stWeeklySched.nSet +1;
			END_IF
			_i := 100;
		ELSE
			(* start ADS write *)
			_fbWriteProp.bExecute := TRUE;
		END_IF

	100: (* Done *)
		bDone := (nErrorId = BACnet_ERR_NO_ERROR);
		(* release ADS buffer *)
		stBACnet_AdsBuffer.iLocked := 0;
		(* release data array *)
		stWeeklySched.bBusy := FALSE;
		(* go idle *)
		_i := 0;

END_CASE

(* set error flag *)
bError 	:= nErrorId > BACnet_ERR_NO_ERROR;
bBusy 	:= _i > 0;
END_FUNCTION_BLOCK
ACTION _NextDay:
_bNextDay := ((_pDailySched^.nEntrySize AND 16#80000000) = 16#80000000);
_cbTmpSize := _F_BACnet_AlignedSize(_pDailySched^.nEntrySize AND 16#7FFFFFFF) + SIZEOF(_pDailySched^.nEntrySize) + SIZEOF(_pDailySched^.nRes);
_pDailySched := _pDailySched + _cbTmpSize;
_cbTotalBuf := _cbTotalBuf + _cbTmpSize;
_pOldTimeValue := 0;
END_ACTION
ACTION _NextTimeValue:
_bNextTimeValue := (_pTimeValue^.nEntrySize AND 16#80000000) = 16#80000000;
_cbTmpSize := _F_BACnet_AlignedSize(_pTimeValue^.nEntrySize AND 16#7FFFFFFF) + SIZEOF(_pDailySched^.stListEntry.nEntrySize) + SIZEOF(_pDailySched^.stListEntry.nRes);
_pOldTimeValue := _pTimeValue;
_pTimeValue := _pTimeValue + _cbTmpSize;
END_ACTION
